TYPE U_Data :
UNION
	sData : STRING(255);
	aData : ARRAY[0..255] OF BYTE;
END_UNION
END_TYPE

(* stored: Version 1.1.0.1, ProductVersion 3.1.4019.2
   DUT U_Data: Id {61532652-25bb-441d-ab1c-8fec28a197c0} *)
